FUNCTION_BLOCK FB_Blink
VAR_INPUT
END_VAR
VAR_OUTPUT
	Fast:BOOL;
	Normal:BOOL;
	Slow:BOOL;
END_VAR
VAR
	TFast:TON;
	TNormal:TON;
	TSlow:TON;

END_VAR

TFast(IN:=NOT TFast.Q , PT:=T#0.1S);
TNormal(IN:=NOT TNormal.Q , PT:=T#0.2S);
TSlow(IN:=NOT TSlow.Q , PT:=T#0.3S);

IF TFast.Q THEN
	(*Toggle bit*)
	Fast:=NOT Fast;
END_IF

IF TNormal.Q THEN
	(*Toggle bit*)
	Normal:=NOT Normal;
END_IF

IF TSlow.Q THEN
	(*Toggle bit*)
	Slow:=NOT Slow;
END_IF

END_FUNCTION_BLOCK

(* stored: Version 1.1.0.1, ProductVersion 3.1.4020.12
   POU FB_Blink: Id {d5e72600-e711-44bf-9f5b-c26d8b84b277}, SpecialFunc None *)
